{attribute 'GeneratedUsingTerminal: EL3773-0000-0016'}
{attribute addProperty BoxType "EL3773-0000-0016"}
{attribute addProperty Id "U3_SAMPLESAT %I*U3_SAMPLES_2D13B74B20"}
{attribute addProperty CRC "3401807246"}
{attribute addProperty Size "20"}
TYPE L3_Voltage_Samples_CAC3758E EXTENDS InputBase_8311D824 :
STRUCT
	{attribute addProperty Name "U3_SAMPLES"}
	U3_SAMPLES AT %I* : U3_SAMPLES_2D13B74B;
END_STRUCT
END_TYPE

(* stored: Version 1.2.0.0, ProductVersion 3.1.4024.9
   DUT L3_Voltage_Samples_CAC3758E: Id {95f227b9-b333-44a1-85eb-ef70529116f0} *)
